KUKA KRL data list: ps_a_lta_res_c02.dat

&ACCESS RVO1
&COMMENT Solda Atego LTA
&PARAM DISKPATH = KRC:\R1\Program\OLP
DEFDAT ps_a_lta_res_c02
;FOLD EXTERNAL DECLARATIONS;%{PE}%MKUKATPBASIS,%CEXT,%VCOMMON,%P
;FOLD GRIPPERTECH EXT
EXT  H50 (INT  :IN,INT  :IN,INT  :IN,GRP_TYP  :IN )
;ENDFOLD (GRIPPERTECH EXT)
;FOLD SPOTTECH EXT
EXT  USERSPOT (S_COMMAND  :IN,SPOT_TYPE  :IN )
;ENDFOLD (SPOTTECH EXT)
;FOLD BASISTECH EXT;%{PE}%MKUKATPBASIS,%CEXT,%VEXT,%P
EXT  BAS (BAS_COMMAND  :IN,REAL  :IN )
DECL INT SUCCESS
;ENDFOLD (BASISTECH EXT)
;FOLD USER EXT;%{E}%MKUKATPUSER,%CEXT,%VEXT,%P
;Make your modifications here

;ENDFOLD (USER EXT)
;ENDFOLD (EXTERNAL DECLARATIONS)
DECL FDAT Fl010={TOOL_NO 3,BASE_NO 3,IPO_FRAME #BASE,POINT2[] " "}
DECL E6POS Xl010={X 137.790894,Y 755.423828,Z 801.72998,A 158.771606,B 69.1498032,C 162.299606,S 18,T 42,E1 0.0,E2 0.0,E3 0.0,E4 0.0,E5 0.0,E6 0.0}
DECL LDAT LL_OLP2={VEL 2.0,ACC 100.0,APO_DIST 10.0,APO_FAC 0.0,ORI_TYP #VAR,CIRC_TYP #BASE,JERK_FAC 50.0}
DECL FDAT Fl015={TOOL_NO 3,BASE_NO 3,IPO_FRAME #BASE,POINT2[] " "}
DECL E6POS Xl015={X 603.140991,Y 808.36499,Z 1241.97498,A 158.485001,B 12.9363003,C 166.735794,S 2,T 42}
DECL LDAT LL_OLP3={VEL 2.0,ACC 100.0,APO_DIST 10.0,APO_FAC 0.0,ORI_TYP #VAR,CIRC_TYP #BASE,JERK_FAC 50.0}
DECL FDAT Fl020={TOOL_NO 3,BASE_NO 3,IPO_FRAME #BASE,POINT2[] " "}
DECL E6POS Xl020={X 583.611084,Y 712.594788,Z 1181.354,A 154.968796,B 9.37294292,C 157.367905,S 18,T 42,E1 0.0,E2 0.0,E3 0.0,E4 0.0,E5 0.0,E6 0.0}
DECL LDAT LL_OLP4={VEL 2.0,ACC 100.0,APO_DIST 10.0,APO_FAC 0.0,ORI_TYP #VAR,CIRC_TYP #BASE,JERK_FAC 50.0}
DECL FDAT Fl025={TOOL_NO 3,BASE_NO 3,IPO_FRAME #BASE,POINT2[] " "}
DECL E6POS Xl025={X 570.496277,Y 697.463013,Z 1145.79199,A 154.968597,B 9.37284756,C 147.3685,S 18,T 42,E1 0.0,E2 0.0,E3 0.0,E4 0.0,E5 0.0,E6 0.0}
DECL LDAT LL_OLP5={VEL 2.0,ACC 100.0,APO_DIST 10.0,APO_FAC 0.0,ORI_TYP #VAR,CIRC_TYP #BASE,JERK_FAC 50.0}
DECL FDAT Fl030={TOOL_NO 3,BASE_NO 3,IPO_FRAME #BASE,POINT2[] " "}
DECL E6POS Xl030={X 582.752014,Y 1585.71301,Z 1144.11096,A 154.969406,B 9.37310028,C 157.3685,S 2,T 42}
DECL LDAT LL_OLP6={VEL 2.0,ACC 100.0,APO_DIST 10.0,APO_FAC 0.0,ORI_TYP #VAR,CIRC_TYP #BASE,JERK_FAC 50.0}
DECL FDAT Fl035={TOOL_NO 3,BASE_NO 3,IPO_FRAME #BASE,POINT2[] " "}
DECL E6POS Xl035={X 897.794006,Y 1320.91504,Z 1221.96802,A -149.936798,B -80.7937012,C 61.0237007,S 2,T 34}
DECL LDAT LL_OLP7={VEL 2.0,ACC 100.0,APO_DIST 30.0,APO_FAC 0.0,ORI_TYP #VAR,CIRC_TYP #BASE,JERK_FAC 50.0}
DECL FDAT Fl040={TOOL_NO 3,BASE_NO 3,IPO_FRAME #BASE,POINT2[] " "}
DECL E6POS Xl040={X 637.291992,Y 987.916992,Z 1221.96594,A -149.936798,B -80.7937012,C 61.0236015,S 2,T 34}
DECL LDAT LL_OLP8={VEL 2.0,ACC 100.0,APO_DIST 2.0,APO_FAC 0.0,ORI_TYP #VAR,CIRC_TYP #BASE,JERK_FAC 50.0}
DECL FDAT Fl045={TOOL_NO 3,BASE_NO 3,IPO_FRAME #BASE,POINT2[] " "}
DECL E6POS Xl045={X 597.394775,Y 971.886719,Z 1312.26404,A -116.101997,B -85.0568771,C 22.43223,S 18,T 34,E1 0.0,E2 0.0,E3 0.0,E4 0.0,E5 0.0,E6 0.0}
DECL LDAT LL_OLP9={VEL 2.0,ACC 100.0,APO_DIST 0.0,APO_FAC 0.0,ORI_TYP #VAR,CIRC_TYP #BASE,JERK_FAC 50.0}
DECL FDAT FSWP_60_9580={TOOL_NO 3,BASE_NO 3,IPO_FRAME #BASE,POINT2[] " "}
DECL E6POS XSWP_60_9580={X 594.554016,Y 986.326416,Z 1318.20105,A -158.479599,B -86.959137,C 65.2630081,S 18,T 34,E1 0.0,E2 0.0,E3 0.0,E4 0.0,E5 0.0,E6 0.0}
DECL LDAT LL_OLP10={VEL 2.0,ACC 100.0,APO_DIST 0.0,APO_FAC 0.0,ORI_TYP #VAR,CIRC_TYP #BASE,JERK_FAC 50.0}
DECL FDAT FSWP_60_9578={TOOL_NO 3,BASE_NO 3,IPO_FRAME #BASE,POINT2[] " "}
DECL E6POS XSWP_60_9578={X 622.752625,Y 986.4104,Z 1319.24805,A 140.785599,B -87.346962,C 128.905701,S 18,T 34,E1 0.0,E2 0.0,E3 0.0,E4 0.0,E5 0.0,E6 0.0}
DECL LDAT LL_OLP11={VEL 2.0,ACC 100.0,APO_DIST 0.0,APO_FAC 0.0,ORI_TYP #VAR,CIRC_TYP #BASE,JERK_FAC 50.0}
DECL FDAT FSWP_60_9590={TOOL_NO 3,BASE_NO 3,IPO_FRAME #BASE,POINT2[] " "}
DECL E6POS XSWP_60_9590={X 649.854675,Y 985.826782,Z 1320.13501,A 149.641907,B -87.5714569,C 121.5755,S 18,T 34,E1 0.0,E2 0.0,E3 0.0,E4 0.0,E5 0.0,E6 0.0}
DECL LDAT LL_OLP12={VEL 2.0,ACC 100.0,APO_DIST 0.0,APO_FAC 0.0,ORI_TYP #VAR,CIRC_TYP #BASE,JERK_FAC 50.0}
DECL FDAT Fl050={TOOL_NO 3,BASE_NO 3,IPO_FRAME #BASE,POINT2[] " "}
DECL E6POS Xl050={X 660.460388,Y 983.00177,Z 1317.37402,A -113.609398,B -85.0964127,C 24.9298801,S 18,T 34,E1 0.0,E2 0.0,E3 0.0,E4 0.0,E5 0.0,E6 0.0}
DECL LDAT LL_OLP13={VEL 2.0,ACC 100.0,APO_DIST 2.0,APO_FAC 0.0,ORI_TYP #VAR,CIRC_TYP #BASE,JERK_FAC 50.0}
DECL FDAT Fl060={TOOL_NO 3,BASE_NO 3,IPO_FRAME #BASE,POINT2[] " ",TQ_STATE FALSE}
DECL E6POS Xl060={X 1323.354,Y 1352.35901,Z 35.526001,A 180.0,B -37.3134003,C 90.0,S 2,T 34}
DECL LDAT LL_OLP15={VEL 2.0,ACC 100.0,APO_DIST 30.0,APO_FAC 0.0,ORI_TYP #VAR,CIRC_TYP #BASE,JERK_FAC 50.0}
DECL FDAT Fl065={TOOL_NO 3,BASE_NO 3,IPO_FRAME #BASE,POINT2[] " "}
DECL E6POS Xl065={X 1312.10205,Y 1148.0,Z 79.7080002,A 180.0,B -13.3133001,C 90.0,S 2,T 42}
DECL FDAT Fl070={TOOL_NO 3,BASE_NO 3,IPO_FRAME #BASE,POINT2[] " ",TQ_STATE FALSE}
DECL E6POS Xl070={X 1116.63403,Y 1017.16602,Z 51.4317093,A 179.996597,B -13.3109398,C 90.0032806,S 18,T 42,E1 0.0,E2 0.0,E3 0.0,E4 0.0,E5 0.0,E6 0.0}
DECL LDAT LL_OLP17={VEL 2.0,ACC 100.0,APO_DIST 5.0,APO_FAC 0.0,ORI_TYP #VAR,CIRC_TYP #BASE,JERK_FAC 50.0}
DECL FDAT Fl075={TOOL_NO 3,BASE_NO 3,IPO_FRAME #BASE,POINT2[] " "}
DECL E6POS Xl075={X 1319.16394,Y 1023.46899,Z 111.884102,A 179.976395,B -22.2574997,C 89.995903,S 18,T 34,E1 0.0,E2 0.0,E3 0.0,E4 0.0,E5 0.0,E6 0.0}
DECL LDAT LL_OLP18={VEL 2.0,ACC 100.0,APO_DIST 0.0,APO_FAC 0.0,ORI_TYP #VAR,CIRC_TYP #BASE,JERK_FAC 50.0}
DECL FDAT FSWP_60_9532={TOOL_NO 3,BASE_NO 3,IPO_FRAME #BASE,POINT2[] " "}
DECL E6POS XSWP_60_9532={X 1309.97205,Y 1033.255,Z 113.483902,A 178.891602,B -22.3080006,C 91.5146637,S 18,T 34,E1 0.0,E2 0.0,E3 0.0,E4 0.0,E5 0.0,E6 0.0}
DECL LDAT LL_OLP19={VEL 2.0,ACC 100.0,APO_DIST 0.0,APO_FAC 0.0,ORI_TYP #VAR,CIRC_TYP #BASE,JERK_FAC 50.0}
DECL FDAT FSWP_60_9530={TOOL_NO 3,BASE_NO 3,IPO_FRAME #BASE,POINT2[] " "}
DECL E6POS XSWP_60_9530={X 1350.33398,Y 1031.08301,Z 116.934502,A 179.234802,B -22.3540192,C 92.9899292,S 18,T 34,E1 0.0,E2 0.0,E3 0.0,E4 0.0,E5 0.0,E6 0.0}
DECL LDAT LL_OLP20={VEL 2.0,ACC 100.0,APO_DIST 0.0,APO_FAC 0.0,ORI_TYP #VAR,CIRC_TYP #BASE,JERK_FAC 50.0}
DECL FDAT FSWP_60_9528={TOOL_NO 3,BASE_NO 3,IPO_FRAME #BASE,POINT2[] " "}
DECL E6POS XSWP_60_9528={X 1398.21704,Y 1031.49902,Z 114.7854,A 178.992905,B -22.3614101,C 93.3113708,S 18,T 34,E1 0.0,E2 0.0,E3 0.0,E4 0.0,E5 0.0,E6 0.0}
DECL LDAT LL_OLP21={VEL 2.0,ACC 100.0,APO_DIST 0.0,APO_FAC 0.0,ORI_TYP #VAR,CIRC_TYP #BASE,JERK_FAC 50.0}
DECL FDAT Fl080={TOOL_NO 3,BASE_NO 3,IPO_FRAME #BASE,POINT2[] " "}
DECL E6POS Xl080={X 1417.18701,Y 1021.49597,Z 96.9904327,A 179.976395,B -22.3135891,C 89.9944611,S 18,T 34,E1 0.0,E2 0.0,E3 0.0,E4 0.0,E5 0.0,E6 0.0}
DECL LDAT LL_OLP22={VEL 2.0,ACC 100.0,APO_DIST 3.0,APO_FAC 0.0,ORI_TYP #VAR,CIRC_TYP #BASE,JERK_FAC 50.0}
DECL FDAT Fl085={TOOL_NO 3,BASE_NO 3,IPO_FRAME #BASE,POINT2[] " ",TQ_STATE FALSE}
DECL E6POS Xl085={X 1438.52002,Y 1019.47498,Z 108.884697,A 179.9823,B -21.8121204,C 91.8203812,S 18,T 34,E1 0.0,E2 0.0,E3 0.0,E4 0.0,E5 0.0,E6 0.0}
DECL LDAT LL_OLP23={VEL 2.0,ACC 100.0,APO_DIST 3.0,APO_FAC 0.0,ORI_TYP #VAR,CIRC_TYP #BASE,JERK_FAC 50.0}
DECL FDAT FSWP_60_9524={TOOL_NO 3,BASE_NO 3,IPO_FRAME #BASE,POINT2[] " "}
DECL E6POS XSWP_60_9524={X 1471.48499,Y 1028.17505,Z 118.2313,A 179.984207,B -21.8108406,C 94.6465912,S 18,T 42,E1 0.0,E2 0.0,E3 0.0,E4 0.0,E5 0.0,E6 0.0}
DECL LDAT LL_OLP24={VEL 2.0,ACC 100.0,APO_DIST 0.0,APO_FAC 0.0,ORI_TYP #VAR,CIRC_TYP #BASE,JERK_FAC 50.0}
DECL FDAT FSWP_60_9522={TOOL_NO 3,BASE_NO 3,IPO_FRAME #BASE,POINT2[] " "}
DECL E6POS XSWP_60_9522={X 1510.82202,Y 1027.48901,Z 117.052101,A 179.633301,B -21.8348503,C 95.0433273,S 18,T 42,E1 0.0,E2 0.0,E3 0.0,E4 0.0,E5 0.0,E6 0.0}
DECL LDAT LL_OLP25={VEL 2.0,ACC 100.0,APO_DIST 0.0,APO_FAC 0.0,ORI_TYP #VAR,CIRC_TYP #BASE,JERK_FAC 50.0}
DECL FDAT FSWP_60_9520={TOOL_NO 3,BASE_NO 3,IPO_FRAME #BASE,POINT2[] " "}
DECL E6POS XSWP_60_9520={X 1561.91602,Y 1025.35901,Z 114.752197,A 179.415298,B -21.8551006,C 95.513092,S 18,T 42,E1 0.0,E2 0.0,E3 0.0,E4 0.0,E5 0.0,E6 0.0}
DECL LDAT LL_OLP26={VEL 2.0,ACC 100.0,APO_DIST 0.0,APO_FAC 0.0,ORI_TYP #VAR,CIRC_TYP #BASE,JERK_FAC 50.0}
DECL FDAT FSWP_60_9516={TOOL_NO 3,BASE_NO 3,IPO_FRAME #BASE,POINT2[] " "}
DECL E6POS XSWP_60_9516={X 1634.89197,Y 1024.49402,Z 113.019402,A 179.995407,B -21.8119507,C 93.8479233,S 18,T 42,E1 0.0,E2 0.0,E3 0.0,E4 0.0,E5 0.0,E6 0.0}
DECL LDAT LL_OLP29={VEL 2.0,ACC 100.0,APO_DIST 0.0,APO_FAC 0.0,ORI_TYP #VAR,CIRC_TYP #BASE,JERK_FAC 50.0}
DECL FDAT FSWP_60_9514={TOOL_NO 3,BASE_NO 3,IPO_FRAME #BASE,POINT2[] " "}
DECL E6POS XSWP_60_9514={X 1684.01099,Y 1024.66504,Z 111.075897,A -179.909302,B -21.8068295,C 94.0637131,S 18,T 42,E1 0.0,E2 0.0,E3 0.0,E4 0.0,E5 0.0,E6 0.0}
DECL LDAT LL_OLP30={VEL 2.0,ACC 100.0,APO_DIST 0.0,APO_FAC 0.0,ORI_TYP #VAR,CIRC_TYP #BASE,JERK_FAC 50.0}
DECL FDAT FSWP_60_9512={TOOL_NO 3,BASE_NO 3,IPO_FRAME #BASE,POINT2[] " "}
DECL E6POS XSWP_60_9512={X 1730.85803,Y 1023.92499,Z 109.979797,A 179.977798,B -21.8196297,C 94.0500793,S 18,T 34,E1 0.0,E2 0.0,E3 0.0,E4 0.0,E5 0.0,E6 0.0}
DECL LDAT LL_OLP31={VEL 2.0,ACC 100.0,APO_DIST 0.0,APO_FAC 0.0,ORI_TYP #VAR,CIRC_TYP #BASE,JERK_FAC 50.0}
DECL FDAT FSWP_60_9510={TOOL_NO 3,BASE_NO 3,IPO_FRAME #BASE,POINT2[] " "}
DECL E6POS XSWP_60_9510={X 1781.72998,Y 1023.367,Z 108.454002,A 179.940598,B -21.8236008,C 94.0563507,S 18,T 34,E1 0.0,E2 0.0,E3 0.0,E4 0.0,E5 0.0,E6 0.0}
DECL LDAT LL_OLP32={VEL 2.0,ACC 100.0,APO_DIST 0.0,APO_FAC 0.0,ORI_TYP #VAR,CIRC_TYP #BASE,JERK_FAC 50.0}
DECL FDAT FSWP_60_9508={TOOL_NO 3,BASE_NO 3,IPO_FRAME #BASE,POINT2[] " "}
DECL E6POS XSWP_60_9508={X 1830.94995,Y 1023.06897,Z 107.122398,A -179.631393,B -21.7844906,C 93.638443,S 18,T 34,E1 0.0,E2 0.0,E3 0.0,E4 0.0,E5 0.0,E6 0.0}
DECL LDAT LL_OLP33={VEL 2.0,ACC 100.0,APO_DIST 0.0,APO_FAC 0.0,ORI_TYP #VAR,CIRC_TYP #BASE,JERK_FAC 50.0}
DECL FDAT FSWP_60_9504={TOOL_NO 3,BASE_NO 3,IPO_FRAME #BASE,POINT2[] " "}
DECL E6POS XSWP_60_9504={X 1931.47095,Y 1021.03998,Z 104.680901,A 179.644196,B -21.8454208,C 91.821701,S 18,T 34,E1 0.0,E2 0.0,E3 0.0,E4 0.0,E5 0.0,E6 0.0}
DECL LDAT LL_OLP34={VEL 2.0,ACC 100.0,APO_DIST 0.0,APO_FAC 0.0,ORI_TYP #VAR,CIRC_TYP #BASE,JERK_FAC 50.0}
DECL FDAT FSWP_60_9502={TOOL_NO 3,BASE_NO 3,IPO_FRAME #BASE,POINT2[] " "}
DECL E6POS XSWP_60_9502={X 1983.68103,Y 1020.96802,Z 103.441002,A 179.871902,B -21.8300705,C 91.4060669,S 18,T 34,E1 0.0,E2 0.0,E3 0.0,E4 0.0,E5 0.0,E6 0.0}
DECL LDAT LL_OLP35={VEL 2.0,ACC 100.0,APO_DIST 0.0,APO_FAC 0.0,ORI_TYP #VAR,CIRC_TYP #BASE,JERK_FAC 50.0}
DECL FDAT FSWP_60_9500={TOOL_NO 3,BASE_NO 3,IPO_FRAME #BASE,POINT2[] " "}
DECL E6POS XSWP_60_9500={X 2031.73096,Y 1020.23798,Z 101.461601,A -179.601303,B -21.6593494,C 93.2189102,S 18,T 34,E1 0.0,E2 0.0,E3 0.0,E4 0.0,E5 0.0,E6 0.0}
DECL LDAT LL_OLP36={VEL 2.0,ACC 100.0,APO_DIST 0.0,APO_FAC 0.0,ORI_TYP #VAR,CIRC_TYP #BASE,JERK_FAC 50.0}
DECL FDAT FSWP_60_9498={TOOL_NO 3,BASE_NO 3,IPO_FRAME #BASE,POINT2[] " "}
DECL E6POS XSWP_60_9498={X 2087.20093,Y 1019.17798,Z 100.790497,A -179.538605,B -24.3359203,C 91.086937,S 18,T 34,E1 0.0,E2 0.0,E3 0.0,E4 0.0,E5 0.0,E6 0.0}
DECL LDAT LL_OLP37={VEL 2.0,ACC 100.0,APO_DIST 0.0,APO_FAC 0.0,ORI_TYP #VAR,CIRC_TYP #BASE,JERK_FAC 50.0}
DECL FDAT FSWP_60_9496={TOOL_NO 3,BASE_NO 3,IPO_FRAME #BASE,POINT2[] " "}
DECL E6POS XSWP_60_9496={X 2153.36206,Y 1017.86603,Z 97.8585434,A -179.961594,B -38.2697296,C 90.7052078,S 18,T 34,E1 0.0,E2 0.0,E3 0.0,E4 0.0,E5 0.0,E6 0.0}
DECL LDAT LL_OLP38={VEL 2.0,ACC 100.0,APO_DIST 0.0,APO_FAC 0.0,ORI_TYP #VAR,CIRC_TYP #BASE,JERK_FAC 50.0}
DECL FDAT Fl100={TOOL_NO 3,BASE_NO 3,IPO_FRAME #BASE,POINT2[] " "}
DECL E6POS Xl100={X 2124.13599,Y 1014.198,Z 40.5825882,A 179.976501,B -21.8289909,C 91.8177567,S 18,T 34,E1 0.0,E2 0.0,E3 0.0,E4 0.0,E5 0.0,E6 0.0}
DECL LDAT LL_OLP39={VEL 2.0,ACC 100.0,APO_DIST 5.0,APO_FAC 0.0,ORI_TYP #VAR,CIRC_TYP #BASE,JERK_FAC 50.0}
DECL FDAT Fl105={TOOL_NO 3,BASE_NO 3,IPO_FRAME #BASE,POINT2[] " "}
DECL E6POS Xl105={X 1973.10205,Y 1113.71301,Z 22.7551403,A -177.173203,B -26.8758907,C 89.4126968,S 18,T 34,E1 0.0,E2 0.0,E3 0.0,E4 0.0,E5 0.0,E6 0.0}
DECL LDAT LL_OLP40={VEL 2.0,ACC 100.0,APO_DIST 30.0,APO_FAC 0.0,ORI_TYP #VAR,CIRC_TYP #BASE,JERK_FAC 50.0}
DECL FDAT Fl110={TOOL_NO 3,BASE_NO 3,IPO_FRAME #BASE,POINT2[] " "}
DECL E6POS Xl110={X 1765.68298,Y 1252.62695,Z 49.1746597,A -178.002701,B -30.1959591,C 89.5175018,S 18,T 34,E1 0.0,E2 0.0,E3 0.0,E4 0.0,E5 0.0,E6 0.0}
DECL FDAT Fl115={TOOL_NO 3,BASE_NO 3,IPO_FRAME #BASE,POINT2[] " "}
DECL PDAT PP_OLP2={VEL 100.0,ACC 100.0,APO_DIST 100.0,APO_MODE #CDIS}
DECL E6POS Xl115={X 1738.02795,Y 2276.4519,Z 99.2014771,A 178.272095,B -17.5484295,C 90.5386963,S 18,T 42,E1 0.0,E2 0.0,E3 0.0,E4 0.0,E5 0.0,E6 0.0}
DECL BASIS_SUGG_T LAST_BASIS={POINT1[] "P10                     ",POINT2[] "P10                     ",CP_PARAMS[] "CPDAT15                 ",PTP_PARAMS[] "PDAT0                   ",CONT[] "C_DIS C_DIS             ",CP_VEL[] "2                       ",PTP_VEL[] "100                     ",SYNC_PARAMS[] "SYNCDAT                 ",SPL_NAME[] "S0                      "}
DECL E6POS XSWP_60_9790={X 724.02002,Y 987.601013,Z 1322.13,A 6.37466097,B -75.1279068,C -93.6373672,S 18,T 34,E1 0.0,E2 0.0,E3 0.0,E4 0.0,E5 0.0,E6 0.0}

DECL FDAT FSWP_60_9790={TOOL_NO 3,BASE_NO 3,IPO_FRAME #BASE,POINT2[] " "}

DECL E6POS XSWP_60_9792={X 760.697815,Y 987.15448,Z 1322.12805,A 4.15385294,B -75.2733917,C -92.2330627,S 18,T 34,E1 0.0,E2 0.0,E3 0.0,E4 0.0,E5 0.0,E6 0.0}

DECL FDAT FSWP_60_9792={TOOL_NO 3,BASE_NO 3,IPO_FRAME #BASE,POINT2[] " "}

DECL E6POS XSWP_60_9794={X 801.021729,Y 987.831726,Z 1322.09094,A 3.81046605,B -75.294632,C -91.246727,S 18,T 34,E1 0.0,E2 0.0,E3 0.0,E4 0.0,E5 0.0,E6 0.0}

DECL FDAT FSWP_60_9794={TOOL_NO 3,BASE_NO 3,IPO_FRAME #BASE,POINT2[] " "}

DECL E6POS XSWP_60_9796={X 847.215515,Y 988.473877,Z 1322.84302,A -7.95260715,B -75.2147827,C -79.8678207,S 18,T 34,E1 0.0,E2 0.0,E3 0.0,E4 0.0,E5 0.0,E6 0.0}

DECL FDAT FSWP_60_9796={TOOL_NO 3,BASE_NO 3,IPO_FRAME #BASE,POINT2[] " "}


DECL E6POS XSWP_60_9798={X 903.10553,Y 988.90387,Z 1322.88794,A -5.96380901,B -75.1801071,C -82.0746765,S 18,T 34,E1 0.0,E2 0.0,E3 0.0,E4 0.0,E5 0.0,E6 0.0}
DECL FDAT FSWP_60_9798={TOOL_NO 3,BASE_NO 3,IPO_FRAME #BASE,POINT2[] " "}

DECL E6POS XSWP_60_9802={X 1004.96802,Y 990.117188,Z 1321.85095,A -9.19126225,B -74.9905014,C -78.2747421,S 18,T 34,E1 0.0,E2 0.0,E3 0.0,E4 0.0,E5 0.0,E6 0.0}

DECL FDAT FSWP_60_9802={TOOL_NO 3,BASE_NO 3,IPO_FRAME #BASE,POINT2[] " "}

DECL E6POS XSWP_60_9804={X 1056.15295,Y 989.565613,Z 1321.62402,A -8.10820961,B -74.9925537,C -79.3390274,S 18,T 34,E1 0.0,E2 0.0,E3 0.0,E4 0.0,E5 0.0,E6 0.0}

DECL FDAT FSWP_60_9804={TOOL_NO 3,BASE_NO 3,IPO_FRAME #BASE,POINT2[] " "}


DECL E6POS XSWP_60_9806={X 1105.53503,Y 989.208618,Z 1321.96997,A -11.5188503,B -74.7813568,C -76.1085663,S 18,T 34,E1 0.0,E2 0.0,E3 0.0,E4 0.0,E5 0.0,E6 0.0}
DECL FDAT FSWP_60_9806={TOOL_NO 3,BASE_NO 3,IPO_FRAME #BASE,POINT2[] " "}
DECL E6POS XSWP_60_9808={X 1144.06299,Y 989.556213,Z 1320.54797,A -9.90100574,B -74.9102707,C -77.5595322,S 18,T 34,E1 0.0,E2 0.0,E3 0.0,E4 0.0,E5 0.0,E6 0.0}
DECL FDAT FSWP_60_9808={TOOL_NO 3,BASE_NO 3,IPO_FRAME #BASE,POINT2[] " "}

DECL E6POS XSWP_60_9810={X 1183.93701,Y 988.581177,Z 1319.66003,A -3.22944999,B -75.0367966,C -84.5192337,S 18,T 34,E1 0.0,E2 0.0,E3 0.0,E4 0.0,E5 0.0,E6 0.0}
DECL FDAT FSWP_60_9810={TOOL_NO 3,BASE_NO 3,IPO_FRAME #BASE,POINT2[] " "}
DECL PDAT PP_OLP4={VEL 100.0,ACC 100.0,APO_DIST 30.0,APO_MODE #CDIS}
DECL E6POS Xl006={X 1083.797,Y 1451.30701,Z 836.236023,A 174.173294,B -30.1965008,C 118.184799,S 2,T 42}
DECL FDAT Fl006={TOOL_NO 3,BASE_NO 3,IPO_FRAME #BASE,POINT2[] " "}
DECL LDAT LL_OLP48={VEL 2.0,ACC 100.0,APO_DIST 30.0,APO_FAC 0.0,ORI_TYP #VAR,CIRC_TYP #BASE,JERK_FAC 50.0}
DECL E6POS Xl011={X 563.752014,Y 1566.71301,Z 1132.11096,A 154.969406,B 9.37310028,C 157.3685,S 2,T 42}
DECL FDAT Fl011={TOOL_NO 3,BASE_NO 3,IPO_FRAME #BASE,POINT2[] " "}
DECL LDAT LL_OLP49={VEL 2.0,ACC 100.0,APO_DIST 10.0,APO_FAC 0.0,ORI_TYP #VAR,CIRC_TYP #BASE,JERK_FAC 50.0}
DECL E6POS Xl016={X 562.511414,Y 691.50061,Z 1119.09802,A 154.969101,B 9.37301254,C 147.368195,S 18,T 42,E1 0.0,E2 0.0,E3 0.0,E4 0.0,E5 0.0,E6 0.0}
DECL FDAT Fl016={TOOL_NO 3,BASE_NO 3,IPO_FRAME #BASE,POINT2[] " "}
DECL PDAT PP_OLP5={VEL 100.0,ACC 100.0,APO_DIST 10.0,APO_MODE #CDIS}
DECL E6POS Xl021={X 564.166016,Y 693.661499,Z 1150.06299,A 154.969101,B 9.37302113,C 157.368195,S 18,T 42,E1 0.0,E2 0.0,E3 0.0,E4 0.0,E5 0.0,E6 0.0}
DECL FDAT Fl021={TOOL_NO 3,BASE_NO 3,IPO_FRAME #BASE,POINT2[] " "}
DECL LDAT LL_OLP50={VEL 2.0,ACC 100.0,APO_DIST 10.0,APO_FAC 0.0,ORI_TYP #VAR,CIRC_TYP #BASE,JERK_FAC 50.0}
DECL E6POS Xl026={X 582.596375,Y 789.625122,Z 1163.21899,A 158.486099,B 12.9365396,C 166.737305,S 18,T 42,E1 0.0,E2 0.0,E3 0.0,E4 0.0,E5 0.0,E6 0.0}
DECL FDAT Fl026={TOOL_NO 3,BASE_NO 3,IPO_FRAME #BASE,POINT2[] " "}
DECL LDAT LCPDAT0={VEL 2.0,ACC 100.0,APO_DIST 100.0,APO_FAC 50.0,AXIS_VEL 100.0,AXIS_ACC 100.0,ORI_TYP #VAR,CIRC_TYP #BASE,JERK_FAC 50.0,GEAR_JERK 50.0,EXAX_IGN 0}
DECL E6POS XP0={X 567.326416,Y 409.623993,Z 1234.31702,A 158.465195,B 12.93505,C 166.748199,S 18,T 42,E1 0.0,E2 0.0,E3 0.0,E4 0.0,E5 0.0,E6 0.0}
DECL FDAT FP0={TOOL_NO 3,BASE_NO 3,IPO_FRAME #BASE,POINT2[] " ",TQ_STATE FALSE}
DECL LDAT LCPDAT1={VEL 2.0,ACC 100.0,APO_DIST 100.0,APO_FAC 50.0,AXIS_VEL 100.0,AXIS_ACC 100.0,ORI_TYP #VAR,CIRC_TYP #BASE,JERK_FAC 50.0,GEAR_JERK 50.0,EXAX_IGN 0}
DECL E6POS XP1={X 622.916321,Y 355.254211,Z 1422.57605,A 157.948105,B 12.9317598,C 166.758606,S 18,T 42,E1 0.0,E2 0.0,E3 0.0,E4 0.0,E5 0.0,E6 0.0}
DECL FDAT FP1={TOOL_NO 3,BASE_NO 3,IPO_FRAME #BASE,POINT2[] " ",TQ_STATE FALSE}
DECL LDAT LCPDAT2={VEL 2.0,ACC 100.0,APO_DIST 30.0,APO_FAC 50.0,AXIS_VEL 100.0,AXIS_ACC 100.0,ORI_TYP #VAR,CIRC_TYP #BASE,JERK_FAC 50.0,GEAR_JERK 50.0,EXAX_IGN 0}
DECL E6POS XP2={X 539.093994,Y 258.427307,Z 1367.42297,A 155.131699,B 22.3258801,C 163.030502,S 18,T 42,E1 0.0,E2 0.0,E3 0.0,E4 0.0,E5 0.0,E6 0.0}
DECL FDAT FP2={TOOL_NO 3,BASE_NO 3,IPO_FRAME #BASE,POINT2[] " ",TQ_STATE FALSE}
DECL LDAT LCPDAT3={VEL 2.0,ACC 100.0,APO_DIST 10.0,APO_FAC 50.0,AXIS_VEL 100.0,AXIS_ACC 100.0,ORI_TYP #VAR,CIRC_TYP #BASE,JERK_FAC 50.0,GEAR_JERK 50.0,EXAX_IGN 0}
DECL E6POS XP3={X 400.828705,Y 277.572998,Z 1191.0,A 150.367203,B 35.5739708,C 156.604507,S 18,T 42,E1 0.0,E2 0.0,E3 0.0,E4 0.0,E5 0.0,E6 0.0}
DECL FDAT FP3={TOOL_NO 3,BASE_NO 3,IPO_FRAME #BASE,POINT2[] " ",TQ_STATE FALSE}
DECL LDAT LL_OLP51={VEL 2.0,ACC 100.0,APO_DIST 10.0,APO_FAC 0.0,ORI_TYP #VAR,CIRC_TYP #BASE,JERK_FAC 50.0}
DECL E6POS Xl031={X 350.266815,Y 288.423492,Z 1120.07996,A 150.391205,B 43.1624107,C 155.955505,S 18,T 42,E1 0.0,E2 0.0,E3 0.0,E4 0.0,E5 0.0,E6 0.0}
DECL FDAT Fl031={TOOL_NO 3,BASE_NO 3,IPO_FRAME #BASE,POINT2[] " "}
DECL PDAT PP_OLP6={VEL 100.0,ACC 100.0,APO_DIST 0.0,APO_MODE #CDIS}
DECL E6POS Xl036={X 317.7453,Y 296.586395,Z 1050.84399,A 147.642303,B 47.8915787,C 153.828995,S 18,T 42,E1 0.0,E2 0.0,E3 0.0,E4 0.0,E5 0.0,E6 0.0}
DECL FDAT Fl036={TOOL_NO 3,BASE_NO 3,IPO_FRAME #BASE,POINT2[] " "}
DECL PDAT PP_OLP7={VEL 100.0,ACC 100.0,APO_DIST 5.0,APO_MODE #CDIS}
DECL E6POS Xl041={X 102.250198,Y 340.10611,Z 682.652588,A 164.808105,B 79.9921112,C 167.133606,S 18,T 42,E1 0.0,E2 0.0,E3 0.0,E4 0.0,E5 0.0,E6 0.0}
DECL FDAT Fl041={TOOL_NO 3,BASE_NO 3,IPO_FRAME #BASE,POINT2[] " "}
DECL LDAT LL_OLP52={VEL 2.0,ACC 100.0,APO_DIST 5.0,APO_FAC 0.0,ORI_TYP #VAR,CIRC_TYP #BASE,JERK_FAC 50.0}
DECL E6POS Xl046={X 71.2702866,Y 356.045807,Z 624.529419,A 159.397202,B 82.8824234,C 161.778595,S 18,T 42,E1 0.0,E2 0.0,E3 0.0,E4 0.0,E5 0.0,E6 0.0}
DECL FDAT Fl046={TOOL_NO 3,BASE_NO 3,IPO_FRAME #BASE,POINT2[] " "}
DECL LDAT LL_OLP53={VEL 2.0,ACC 100.0,APO_DIST 0.0,APO_FAC 0.0,ORI_TYP #VAR,CIRC_TYP #BASE,JERK_FAC 50.0}
DECL E6POS XSWP_60_7880={X 93.7982178,Y 380.760986,Z 613.06543,A 159.360794,B 82.8838272,C 161.736404,S 18,T 42,E1 0.0,E2 0.0,E3 0.0,E4 0.0,E5 0.0,E6 0.0}
DECL FDAT FSWP_60_7880={TOOL_NO 3,BASE_NO 3,IPO_FRAME #BASE,POINT2[] " "}
DECL LDAT LL_OLP54={VEL 2.0,ACC 100.0,APO_DIST 0.0,APO_FAC 0.0,ORI_TYP #VAR,CIRC_TYP #BASE,JERK_FAC 50.0}
DECL E6POS XSWP_60_7882={X 95.1983414,Y 412.033203,Z 612.224121,A 159.370499,B 82.8822937,C 161.745895,S 18,T 42,E1 0.0,E2 0.0,E3 0.0,E4 0.0,E5 0.0,E6 0.0}
DECL FDAT FSWP_60_7882={TOOL_NO 3,BASE_NO 3,IPO_FRAME #BASE,POINT2[] " "}
DECL LDAT LL_OLP55={VEL 2.0,ACC 100.0,APO_DIST 0.0,APO_FAC 0.0,ORI_TYP #VAR,CIRC_TYP #BASE,JERK_FAC 50.0}
DECL E6POS XSWP_60_7886={X 98.8377228,Y 478.136993,Z 615.090515,A 158.5354,B 82.6687012,C 159.334305,S 18,T 42,E1 0.0,E2 0.0,E3 0.0,E4 0.0,E5 0.0,E6 0.0}
DECL FDAT FSWP_60_7886={TOOL_NO 3,BASE_NO 3,IPO_FRAME #BASE,POINT2[] " "}
DECL LDAT LL_OLP56={VEL 2.0,ACC 100.0,APO_DIST 0.0,APO_FAC 0.0,ORI_TYP #VAR,CIRC_TYP #BASE,JERK_FAC 50.0}
DECL E6POS XSWP_60_7888={X 100.442497,Y 513.4646,Z 616.12793,A 159.082596,B 82.9018936,C 159.794601,S 18,T 42,E1 0.0,E2 0.0,E3 0.0,E4 0.0,E5 0.0,E6 0.0}
DECL FDAT FSWP_60_7888={TOOL_NO 3,BASE_NO 3,IPO_FRAME #BASE,POINT2[] " "}
DECL LDAT LL_OLP57={VEL 2.0,ACC 100.0,APO_DIST 0.0,APO_FAC 0.0,ORI_TYP #VAR,CIRC_TYP #BASE,JERK_FAC 50.0}
DECL E6POS XSWP_60_7890={X 102.522003,Y 545.988403,Z 614.039917,A 160.234299,B 82.879837,C 161.132095,S 18,T 42,E1 0.0,E2 0.0,E3 0.0,E4 0.0,E5 0.0,E6 0.0}
DECL FDAT FSWP_60_7890={TOOL_NO 3,BASE_NO 3,IPO_FRAME #BASE,POINT2[] " "}
DECL LDAT LL_OLP58={VEL 2.0,ACC 100.0,APO_DIST 0.0,APO_FAC 0.0,ORI_TYP #VAR,CIRC_TYP #BASE,JERK_FAC 50.0}
DECL E6POS XSWP_60_7892={X 103.919098,Y 574.488892,Z 615.100891,A 159.7061,B 82.8799286,C 161.684998,S 18,T 42,E1 0.0,E2 0.0,E3 0.0,E4 0.0,E5 0.0,E6 0.0}
DECL FDAT FSWP_60_7892={TOOL_NO 3,BASE_NO 3,IPO_FRAME #BASE,POINT2[] " "}
DECL LDAT LL_OLP59={VEL 2.0,ACC 100.0,APO_DIST 0.0,APO_FAC 0.0,ORI_TYP #VAR,CIRC_TYP #BASE,JERK_FAC 50.0}
DECL E6POS XSWP_60_7896={X 108.416,Y 646.456177,Z 614.435181,A 159.410507,B 82.8830185,C 161.785904,S 18,T 42,E1 0.0,E2 0.0,E3 0.0,E4 0.0,E5 0.0,E6 0.0}
DECL FDAT FSWP_60_7896={TOOL_NO 3,BASE_NO 3,IPO_FRAME #BASE,POINT2[] " "}
DECL LDAT LL_OLP77={VEL 2.0,ACC 100.0,APO_DIST 0.0,APO_FAC 0.0,ORI_TYP #VAR,CIRC_TYP #BASE,JERK_FAC 50.0}
DECL E6POS XSWP_60_7898={X 111.716202,Y 682.766418,Z 615.322815,A 159.398407,B 82.8831482,C 161.775604,S 18,T 42,E1 0.0,E2 0.0,E3 0.0,E4 0.0,E5 0.0,E6 0.0}
DECL FDAT FSWP_60_7898={TOOL_NO 3,BASE_NO 3,IPO_FRAME #BASE,POINT2[] " "}
DECL LDAT LL_OLP78={VEL 2.0,ACC 100.0,APO_DIST 0.0,APO_FAC 0.0,ORI_TYP #VAR,CIRC_TYP #BASE,JERK_FAC 50.0}
DECL E6POS XSWP_60_7900={X 114.766197,Y 718.722412,Z 616.54657,A 159.434402,B 82.8802872,C 161.813995,S 18,T 42,E1 0.0,E2 0.0,E3 0.0,E4 0.0,E5 0.0,E6 0.0}
DECL FDAT FSWP_60_7900={TOOL_NO 3,BASE_NO 3,IPO_FRAME #BASE,POINT2[] " "}
DECL LDAT LL_OLP79={VEL 2.0,ACC 100.0,APO_DIST 0.0,APO_FAC 0.0,ORI_TYP #VAR,CIRC_TYP #BASE,JERK_FAC 50.0}
DECL E6POS XSWP_60_7902={X 119.6847,Y 754.768677,Z 617.763794,A 159.414795,B 82.8860092,C 161.790604,S 18,T 42,E1 0.0,E2 0.0,E3 0.0,E4 0.0,E5 0.0,E6 0.0}
DECL FDAT FSWP_60_7902={TOOL_NO 3,BASE_NO 3,IPO_FRAME #BASE,POINT2[] " "}
DECL LDAT LL_OLP80={VEL 2.0,ACC 100.0,APO_DIST 0.0,APO_FAC 0.0,ORI_TYP #VAR,CIRC_TYP #BASE,JERK_FAC 50.0}
DECL E6POS XSWP_60_7904={X 124.171097,Y 792.095215,Z 620.319885,A 159.417404,B 82.8863602,C 161.792404,S 18,T 42,E1 0.0,E2 0.0,E3 0.0,E4 0.0,E5 0.0,E6 0.0}
DECL FDAT FSWP_60_7904={TOOL_NO 3,BASE_NO 3,IPO_FRAME #BASE,POINT2[] " "}
DECL LDAT LL_OLP81={VEL 2.0,ACC 100.0,APO_DIST 0.0,APO_FAC 0.0,ORI_TYP #VAR,CIRC_TYP #BASE,JERK_FAC 50.0}
DECL E6POS XSWP_60_7906={X 133.554703,Y 847.09137,Z 622.990479,A 158.070801,B 82.8795624,C 162.259598,S 18,T 42,E1 0.0,E2 0.0,E3 0.0,E4 0.0,E5 0.0,E6 0.0}
DECL FDAT FSWP_60_7906={TOOL_NO 3,BASE_NO 3,IPO_FRAME #BASE,POINT2[] " "}
DECL LDAT LL_OLP82={VEL 2.0,ACC 100.0,APO_DIST 0.0,APO_FAC 0.0,ORI_TYP #VAR,CIRC_TYP #BASE,JERK_FAC 50.0}
DECL E6POS XSWP_60_7908={X 139.9673,Y 879.15332,Z 621.591309,A 159.403,B 82.8970566,C 167.299698,S 18,T 42,E1 0.0,E2 0.0,E3 0.0,E4 0.0,E5 0.0,E6 0.0}
DECL FDAT FSWP_60_7908={TOOL_NO 3,BASE_NO 3,IPO_FRAME #BASE,POINT2[] " "}
DECL E6POS Xl051={X 137.945007,Y 854.049988,Z 676.479004,A 164.794098,B 79.9898987,C 167.113907,S 2,T 42,E1 0.0,E2 0.0,E3 0.0,E4 0.0,E5 0.0,E6 0.0}
DECL FDAT Fl051={TOOL_NO 3,BASE_NO 3,IPO_FRAME #BASE,POINT2[] " "}
DECL E6POS XP5={X 420.465912,Y 747.624695,Z 1123.48804,A 158.533401,B 32.2998009,C 165.156693,S 18,T 42,E1 0.0,E2 0.0,E3 0.0,E4 0.0,E5 0.0,E6 0.0}
DECL FDAT FP5={TOOL_NO 3,BASE_NO 3,IPO_FRAME #BASE,POINT2[] " ",TQ_STATE FALSE}
DECL LDAT LCPDAT5={VEL 2.0,ACC 100.0,APO_DIST 10.0,APO_FAC 50.0,AXIS_VEL 100.0,AXIS_ACC 100.0,ORI_TYP #VAR,CIRC_TYP #BASE,JERK_FAC 50.0,GEAR_JERK 50.0,EXAX_IGN 0}
DECL E6POS XP6={X 1011.94702,Y 1316.37695,Z 872.489502,A -166.842194,B -74.2261429,C 77.8371201,S 18,T 34,E1 0.0,E2 0.0,E3 0.0,E4 0.0,E5 0.0,E6 0.0}
DECL FDAT FP6={TOOL_NO 3,BASE_NO 3,IPO_FRAME #BASE,POINT2[] " ",TQ_STATE FALSE}
DECL LDAT LL_OLP83={VEL 2.0,ACC 100.0,APO_DIST 2.0,APO_FAC 0.0,ORI_TYP #VAR,CIRC_TYP #BASE,JERK_FAC 50.0}
DECL E6POS Xl023={X 699.365295,Y 978.134216,Z 1321.15503,A -20.2005806,B -78.3323669,C -68.1035538,S 18,T 34,E1 0.0,E2 0.0,E3 0.0,E4 0.0,E5 0.0,E6 0.0}
DECL FDAT Fl023={TOOL_NO 3,BASE_NO 3,IPO_FRAME #BASE,POINT2[] " "}
DECL LDAT LL_OLP84={VEL 2.0,ACC 100.0,APO_DIST 0.0,APO_FAC 0.0,ORI_TYP #VAR,CIRC_TYP #BASE,JERK_FAC 50.0}
DECL LDAT LL_OLP85={VEL 2.0,ACC 100.0,APO_DIST 0.0,APO_FAC 0.0,ORI_TYP #VAR,CIRC_TYP #BASE,JERK_FAC 50.0}

DECL LDAT LL_OLP86={VEL 2.0,ACC 100.0,APO_DIST 0.0,APO_FAC 0.0,ORI_TYP #VAR,CIRC_TYP #BASE,JERK_FAC 50.0}

DECL LDAT LL_OLP87={VEL 2.0,ACC 100.0,APO_DIST 0.0,APO_FAC 0.0,ORI_TYP #VAR,CIRC_TYP #BASE,JERK_FAC 50.0}
DECL LDAT LL_OLP88={VEL 2.0,ACC 100.0,APO_DIST 0.0,APO_FAC 0.0,ORI_TYP #VAR,CIRC_TYP #BASE,JERK_FAC 50.0}
DECL LDAT LL_OLP89={VEL 2.0,ACC 100.0,APO_DIST 0.0,APO_FAC 0.0,ORI_TYP #VAR,CIRC_TYP #BASE,JERK_FAC 50.0}
DECL LDAT LL_OLP90={VEL 2.0,ACC 100.0,APO_DIST 0.0,APO_FAC 0.0,ORI_TYP #VAR,CIRC_TYP #BASE,JERK_FAC 50.0}
DECL LDAT LL_OLP91={VEL 2.0,ACC 100.0,APO_DIST 0.0,APO_FAC 0.0,ORI_TYP #VAR,CIRC_TYP #BASE,JERK_FAC 50.0}
DECL LDAT LL_OLP92={VEL 2.0,ACC 100.0,APO_DIST 0.0,APO_FAC 0.0,ORI_TYP #VAR,CIRC_TYP #BASE,JERK_FAC 50.0}
DECL LDAT LL_OLP93={VEL 2.0,ACC 100.0,APO_DIST 0.0,APO_FAC 0.0,ORI_TYP #VAR,CIRC_TYP #BASE,JERK_FAC 50.0}
DECL LDAT LL_OLP94={VEL 2.0,ACC 100.0,APO_DIST 0.0,APO_FAC 0.0,ORI_TYP #VAR,CIRC_TYP #BASE,JERK_FAC 50.0}
DECL E6POS Xl028={X 1184.32397,Y 978.322083,Z 1317.11304,A -14.4974499,B -74.4626236,C -73.6468124,S 18,T 34,E1 0.0,E2 0.0,E3 0.0,E4 0.0,E5 0.0,E6 0.0}


DECL FDAT Fl028={TOOL_NO 3,BASE_NO 3,IPO_FRAME #BASE,POINT2[] " "}
DECL LDAT LL_OLP95={VEL 2.0,ACC 100.0,APO_DIST 5.0,APO_FAC 0.0,ORI_TYP #VAR,CIRC_TYP #BASE,JERK_FAC 50.0}
DECL E6POS Xl033={X 1167.98999,Y 981.75531,Z 1261.08606,A -24.1799507,B -79.9280014,C -64.1580505,S 18,T 34,E1 0.0,E2 0.0,E3 0.0,E4 0.0,E5 0.0,E6 0.0}
DECL FDAT Fl033={TOOL_NO 3,BASE_NO 3,IPO_FRAME #BASE,POINT2[] " "}
DECL PDAT PPDAT1={VEL 100.0,ACC 100.0,APO_DIST 30.0,APO_MODE #CDIS,GEAR_JERK 50.0}
DECL E6POS XP7={X 1899.93604,Y 3567.76489,Z 589.863708,A -176.116592,B -26.2018795,C -91.7760925,S 18,T 42,E1 0.0,E2 0.0,E3 0.0,E4 0.0,E5 0.0,E6 0.0}

DECL FDAT FP7={TOOL_NO 4,BASE_NO 3,IPO_FRAME #BASE,POINT2[] " ",TQ_STATE FALSE}
DECL PDAT PPDAT2={VEL 100.0,ACC 100.0,APO_DIST 100.0,APO_MODE #CDIS,GEAR_JERK 50.0}
DECL LDAT LCPDAT7={VEL 2.0,ACC 100.0,APO_DIST 30.0,APO_FAC 50.0,AXIS_VEL 100.0,AXIS_ACC 100.0,ORI_TYP #VAR,CIRC_TYP #BASE,JERK_FAC 50.0,GEAR_JERK 50.0,EXAX_IGN 0}

DECL E6POS XSWP_60_9398={X 2127.0249,Y 1018.26898,Z 99.4095612,A 179.695694,B -26.7392998,C 91.7997437,S 18,T 34,E1 0.0,E2 0.0,E3 0.0,E4 0.0,E5 0.0,E6 0.0}
DECL FDAT FSWP_60_9398={TOOL_NO 3,BASE_NO 3,IPO_FRAME #BASE,POINT2[] " ",TQ_STATE FALSE}
DECL SPOT_SUGG_T LAST_SPOT={GUN[] "2                       ",RETR_CMD[] "#OPN                    ",CHOISE[] "#FIRST                  ",CLO_TM[] "1                       ",PGNO1[] "187                     ",PRESS1[] "0                       ",PGNO2[] "1                       ",PRESS2[] "0                       ",SPOT_PARAMS[] "NORMAL                  "}
DECL SPOT_TYPE SNORMAL={GUN 1,PAIR #FIRST,RETR #OPN,CLO_TM 0,PGNO1 1,PRESS1 0.0,PGNO2 0,PRESS2 0.0}
DECL E6POS XSWP_60_7346={X 145.027603,Y 915.333679,Z 621.085388,A 92.0242233,B 54.5311508,C 101.880501,S 18,T 42,E1 0.0,E2 0.0,E3 0.0,E4 0.0,E5 0.0,E6 0.0}
DECL FDAT FSWP_60_7346={TOOL_NO 3,BASE_NO 3,IPO_FRAME #BASE,POINT2[] " ",TQ_STATE FALSE}
DECL LDAT LCPDAT4={VEL 2.0,ACC 100.0,APO_DIST 100.0,APO_FAC 50.0,AXIS_VEL 100.0,AXIS_ACC 100.0,ORI_TYP #VAR,CIRC_TYP #BASE,JERK_FAC 50.0,GEAR_JERK 50.0,EXAX_IGN 0}
DECL LDAT LCPDAT6={VEL 2.0,ACC 100.0,APO_DIST 10.0,APO_FAC 50.0,AXIS_VEL 100.0,AXIS_ACC 100.0,ORI_TYP #VAR,CIRC_TYP #BASE,JERK_FAC 50.0,GEAR_JERK 50.0,EXAX_IGN 0}
DECL LDAT LCPDAT8={VEL 2.0,ACC 100.0,APO_DIST 30.0,APO_FAC 50.0,AXIS_VEL 100.0,AXIS_ACC 100.0,ORI_TYP #VAR,CIRC_TYP #BASE,JERK_FAC 50.0,GEAR_JERK 50.0,EXAX_IGN 0}
DECL E6POS XP4={X 1230.61096,Y 1015.41901,Z 62.1031799,A -179.999207,B -13.3151903,C 90.0011368,S 18,T 42,E1 0.0,E2 0.0,E3 0.0,E4 0.0,E5 0.0,E6 0.0}
DECL FDAT FP4={TOOL_NO 3,BASE_NO 3,IPO_FRAME #BASE,POINT2[] " ",TQ_STATE FALSE}
DECL LDAT LCPDAT9={VEL 2.0,ACC 100.0,APO_DIST 5.0,APO_FAC 50.0,AXIS_VEL 100.0,AXIS_ACC 100.0,ORI_TYP #VAR,CIRC_TYP #BASE,JERK_FAC 50.0,GEAR_JERK 50.0,EXAX_IGN 0}
DECL E6POS XP8={X 1108.78296,Y 1017.35999,Z 73.2284927,A 179.996597,B -13.3102198,C 90.0024872,S 18,T 42,E1 0.0,E2 0.0,E3 0.0,E4 0.0,E5 0.0,E6 0.0}
DECL FDAT FP8={TOOL_NO 3,BASE_NO 3,IPO_FRAME #BASE,POINT2[] " ",TQ_STATE FALSE}
DECL LDAT LCPDAT10={VEL 2.0,ACC 100.0,APO_DIST 5.0,APO_FAC 50.0,AXIS_VEL 100.0,AXIS_ACC 100.0,ORI_TYP #VAR,CIRC_TYP #BASE,JERK_FAC 50.0,GEAR_JERK 50.0,EXAX_IGN 0}
DECL E6POS XSWP_61_7028={X 1106.75,Y 1027.08203,Z 73.5821381,A 179.582397,B -13.3118801,C 90.0140533,S 18,T 42,E1 0.0,E2 0.0,E3 0.0,E4 0.0,E5 0.0,E6 0.0}
DECL FDAT FSWP_61_7028={TOOL_NO 3,BASE_NO 3,IPO_FRAME #BASE,POINT2[] " ",TQ_STATE FALSE}
DECL LDAT LCPDAT11={VEL 2.0,ACC 100.0,APO_DIST 100.0,APO_FAC 50.0,AXIS_VEL 100.0,AXIS_ACC 100.0,ORI_TYP #VAR,CIRC_TYP #BASE,JERK_FAC 50.0,GEAR_JERK 50.0,EXAX_IGN 0}
DECL E6POS XSWP_61_7030={X 1150.90601,Y 1029.78796,Z 90.5489731,A -179.999695,B -13.3078098,C 90.0062103,S 18,T 42,E1 0.0,E2 0.0,E3 0.0,E4 0.0,E5 0.0,E6 0.0}
DECL FDAT FSWP_61_7030={TOOL_NO 3,BASE_NO 3,IPO_FRAME #BASE,POINT2[] " ",TQ_STATE FALSE}
DECL LDAT LCPDAT12={VEL 2.0,ACC 100.0,APO_DIST 100.0,APO_FAC 50.0,AXIS_VEL 100.0,AXIS_ACC 100.0,ORI_TYP #VAR,CIRC_TYP #BASE,JERK_FAC 50.0,GEAR_JERK 50.0,EXAX_IGN 0}
DECL E6POS XSWP_61_7032={X 1207.87695,Y 1032.18506,Z 98.9621429,A -179.906403,B -19.7675896,C 90.0270386,S 18,T 34,E1 0.0,E2 0.0,E3 0.0,E4 0.0,E5 0.0,E6 0.0}
DECL FDAT FSWP_61_7032={TOOL_NO 3,BASE_NO 3,IPO_FRAME #BASE,POINT2[] " ",TQ_STATE FALSE}
DECL LDAT LCPDAT13={VEL 2.0,ACC 100.0,APO_DIST 100.0,APO_FAC 50.0,AXIS_VEL 100.0,AXIS_ACC 100.0,ORI_TYP #VAR,CIRC_TYP #BASE,JERK_FAC 50.0,GEAR_JERK 50.0,EXAX_IGN 0}
DECL E6POS XP9={X 1206.38403,Y 1006.83502,Z 67.4408493,A -179.908997,B -19.7681408,C 90.0280304,S 18,T 34,E1 0.0,E2 0.0,E3 0.0,E4 0.0,E5 0.0,E6 0.0}
DECL FDAT FP9={TOOL_NO 3,BASE_NO 3,IPO_FRAME #BASE,POINT2[] " ",TQ_STATE FALSE}
DECL LDAT LCPDAT14={VEL 2.0,ACC 100.0,APO_DIST 10.0,APO_FAC 50.0,AXIS_VEL 100.0,AXIS_ACC 100.0,ORI_TYP #VAR,CIRC_TYP #BASE,JERK_FAC 50.0,GEAR_JERK 50.0,EXAX_IGN 0}
DECL E6POS XP10={X 1318.55103,Y 1023.52502,Z 83.9089737,A 179.978394,B -22.2589493,C 89.9975967,S 18,T 34,E1 0.0,E2 0.0,E3 0.0,E4 0.0,E5 0.0,E6 0.0}
DECL FDAT FP10={TOOL_NO 3,BASE_NO 3,IPO_FRAME #BASE,POINT2[] " ",TQ_STATE FALSE}
DECL LDAT LCPDAT15={VEL 2.0,ACC 100.0,APO_DIST 10.0,APO_FAC 50.0,AXIS_VEL 100.0,AXIS_ACC 100.0,ORI_TYP #VAR,CIRC_TYP #BASE,JERK_FAC 50.0,GEAR_JERK 50.0,EXAX_IGN 0}
DECL PDAT PPDAT3={VEL 100.0,ACC 100.0,APO_DIST 0.0,APO_MODE #CDIS,GEAR_JERK 50.0}
ENDDAT
